# B&R Automation Studio project OpcUaSample410_BrbLibUa103 (part 10)

#### BrbUaAddNodeClassText.c - Gibt den Text einer NodeClass zurück
```c
#include <bur/plctypes.h>
#ifdef __cplusplus
	extern "C"
	{
#endif

#include "BrbLibUa.h"
#include <string.h>

#ifdef __cplusplus
	};
#endif

// NOLINTBEGIN(readability-*, bugprone-easily-swappable-parameters, bugprone-branch-clone, clang-diagnostic-invalid-utf8, clang-diagnostic-invalid-source-encoding, clang-diagnostic-pointer-arith, clang-diagnostic-strict-prototypes, hicpp-uppercase-literal-suffix, cppcoreguidelines-*, performance-*)

/* Hängt den Text einer NodeClass an */
plcdword BrbUaAddNodeClassText(enum UANodeClass eNodeClass, plcstring* pText, unsigned long nTextSize)
{
	DWORD nStatus = 0x80460000; // = Bad_StructureMissing
	if(pText != 0)
	{
		nStatus = 0x00000000; // = Good
		switch(eNodeClass)
		{
			case UANodeClass_None:
				BrbStringCat(pText, "None", nTextSize);
				break;

			case UANodeClass_Object:
				BrbStringCat(pText, "Object", nTextSize);
				break;

			case UANodeClass_Variable:
				BrbStringCat(pText, "Variable", nTextSize);
				break;

			case UANodeClass_Method:
				BrbStringCat(pText, "Method", nTextSize);
				break;

			case UANodeClass_ObjectType:
				BrbStringCat(pText, "ObjectType", nTextSize);
				break;

			case UANodeClass_VariableType:
				BrbStringCat(pText, "VariableType", nTextSize);
				break;

			case UANodeClass_ReferenceType:
				BrbStringCat(pText, "ReferenceType", nTextSize);
				break;

			case UANodeClass_DataType:
				BrbStringCat(pText, "DataType", nTextSize);
				break;

			case UANodeClass_View:
				BrbStringCat(pText, "View", nTextSize);
				break;

			case UANodeClass_All:
				BrbStringCat(pText, "All", nTextSize);
				break;

			default: // NOLINT(clang-diagnostic-covered-switch-default)
				BrbStringCat(pText, "Unknown", nTextSize);
				break;

		}
	}
	return nStatus;
}

// NOLINTEND(readability-*, bugprone-easily-swappable-parameters, bugprone-branch-clone, clang-diagnostic-invalid-utf8, clang-diagnostic-invalid-source-encoding, clang-diagnostic-pointer-arith, clang-diagnostic-strict-prototypes, hicpp-uppercase-literal-suffix, cppcoreguidelines-*, performance-*)
```

#### BrbUaAddDatatypeIdText.c - Gibt den Text zu einem Datentyp-Identifier zurück
```c
#include <bur/plctypes.h>
#ifdef __cplusplus
	extern "C"
	{
#endif

#include "BrbLibUa.h"
#include <string.h>

#ifdef __cplusplus
	};
#endif

// NOLINTBEGIN(readability-*, bugprone-easily-swappable-parameters, bugprone-branch-clone, clang-diagnostic-invalid-utf8, clang-diagnostic-invalid-source-encoding, clang-diagnostic-pointer-arith, clang-diagnostic-strict-prototypes, hicpp-uppercase-literal-suffix, cppcoreguidelines-*, performance-*)

/* Hängt den Text zu einem Datentyp-Identifier an */
plcdword BrbUaAddDatatypeIdText(unsigned long nDatatypeId, plcstring* pText, unsigned long nTextSize)
{
	DWORD nStatus = 0x80460000; // = Bad_StructureMissing
	if(pText != 0)
	{
		nStatus = 0x00000000; // = Good
		if(nDatatypeId == 1)
		{
			BrbStringCat(pText, "1=Boolean", nTextSize);
		}
		else if(nDatatypeId == 2)
		{
			BrbStringCat(pText, "2=SByte", nTextSize);
		}
		else if(nDatatypeId == 3)
		{
			BrbStringCat(pText, "3=Byte", nTextSize);
		}
		else if(nDatatypeId == 4)
		{
			BrbStringCat(pText, "4=Int16", nTextSize);
		}
		else if(nDatatypeId == 5)
		{
			BrbStringCat(pText, "5=UInt16", nTextSize);
		}
		else if(nDatatypeId == 6)
		{
			BrbStringCat(pText, "6=Int32", nTextSize);
		}
		else if(nDatatypeId == 7)
		{
			BrbStringCat(pText, "7=UInt32", nTextSize);
		}
		else if(nDatatypeId == 8)
		{
			BrbStringCat(pText, "8=Int64", nTextSize);
		}
		else if(nDatatypeId == 9)
		{
			BrbStringCat(pText, "9=UInt64", nTextSize);
		}
		else if(nDatatypeId == 10)
		{
			BrbStringCat(pText, "10=Float", nTextSize);
		}
		else if(nDatatypeId == 11)
		{
			BrbStringCat(pText, "11=Double", nTextSize);
		}
		else if(nDatatypeId == 12)
		{
			BrbStringCat(pText, "12=String", nTextSize);
		}
		else if(nDatatypeId == 13)
		{
			BrbStringCat(pText, "13=DateTime", nTextSize);
		}
		else if(nDatatypeId == 14)
		{
			BrbStringCat(pText, "14=Guid", nTextSize);
		}
		else if(nDatatypeId == 15)
		{
			BrbStringCat(pText, "15=ByteString", nTextSize);
		}
		else if(nDatatypeId == 16)
		{
			BrbStringCat(pText, "16=XmlElement", nTextSize);
		}
		else if(nDatatypeId == 17)
		{
			BrbStringCat(pText, "17=NodeId", nTextSize);
		}
		else if(nDatatypeId == 18)
		{
			BrbStringCat(pText, "18=ExpandedNodeId", nTextSize);
		}
		else if(nDatatypeId == 19)
		{
			BrbStringCat(pText, "19=StatusCode", nTextSize);
		}
		else if(nDatatypeId == 20)
		{
			BrbStringCat(pText, "20=QualifiedName", nTextSize);
		}
		else if(nDatatypeId == 21)
		{
			BrbStringCat(pText, "21=LocalizedText", nTextSize);
		}
		else if(nDatatypeId == 22)
		{
			BrbStringCat(pText, "22=Structure", nTextSize);
		}
		else if(nDatatypeId == 23)
		{
			BrbStringCat(pText, "23=DataValue", nTextSize);
		}
		else if(nDatatypeId == 25)
		{
			BrbStringCat(pText, "25=DiagnosticInfo", nTextSize);
		}
		else if(nDatatypeId == 26)
		{
			BrbStringCat(pText, "26=Number", nTextSize);
		}
		else if(nDatatypeId == 29)
		{
			BrbStringCat(pText, "29=Enumeration", nTextSize);
		}
		else if(nDatatypeId == 121)
		{
			BrbStringCat(pText, "121=Decimal128", nTextSize);
		}
		else
		{
			STRING sHelp[nBRBUA_VALUE_TEXT_CHAR_MAX];
			BrbUdintToAscii(nDatatypeId, sHelp);
			BrbStringCat(pText, sHelp, nTextSize);
		}
	}
	return nStatus;
}

// NOLINTEND(readability-*, bugprone-easily-swappable-parameters, bugprone-branch-clone, clang-diagnostic-invalid-utf8, clang-diagnostic-invalid-source-encoding, clang-diagnostic-pointer-arith, clang-diagnostic-strict-prototypes, hicpp-uppercase-literal-suffix, cppcoreguidelines-*, performance-*)
```

#### BrbUaAddArrayDimensionText.c - Gibt den Text für eine ArrayDimension zurück
```c
#include <bur/plctypes.h>
#ifdef __cplusplus
	extern "C"
	{
#endif

#include "BrbLibUa.h"
#include <string.h>

#ifdef __cplusplus
	};
#endif

// NOLINTBEGIN(readability-*, bugprone-easily-swappable-parameters, bugprone-branch-clone, clang-diagnostic-invalid-utf8, clang-diagnostic-invalid-source-encoding, clang-diagnostic-pointer-arith, clang-diagnostic-strict-prototypes, hicpp-uppercase-literal-suffix, cppcoreguidelines-*, performance-*)

/* Hängt den Text für eine ArrayDimension an */
plcdword BrbUaAddArrayDimensionText(unsigned long* pArrayDimension, signed long nValueRank, plcstring* pText, unsigned long nTextSize)
{
	DWORD nStatus = 0x80460000; // = Bad_StructureMissing
	if(pArrayDimension != 0 && pText != 0)
	{
		nStatus = 0x800F0000; // = Bad_NothingToDo
		if(nValueRank > 0)
		{
			nStatus = 0x00000000; // = Good
			DINT nIndex = 0;
			STRING sHelp[nBRBUA_VALUE_TEXT_CHAR_MAX];
			if(nValueRank > (DINT)MAX_ELEMENTS_ARRAYDIMENSION)
			{
				nValueRank = MAX_ELEMENTS_ARRAYDIMENSION;
			}
			for(nIndex=0; nIndex<=nValueRank-1; nIndex++)
			{
				UDINT* pDim = ((UDINT*)pArrayDimension) + nIndex;
				BrbUdintToAscii(*pDim, sHelp);
				BrbStringCat(pText, sHelp, nTextSize);
				BrbStringCat(pText, ";", nTextSize);
			}
			BrbStringTrimRight(pText, ";");
		}
	}
	return nStatus;
}

// NOLINTEND(readability-*, bugprone-easily-swappable-parameters, bugprone-branch-clone, clang-diagnostic-invalid-utf8, clang-diagnostic-invalid-source-encoding, clang-diagnostic-pointer-arith, clang-diagnostic-strict-prototypes, hicpp-uppercase-literal-suffix, cppcoreguidelines-*, performance-*)
```

#### BrbUaAddAccessLevelText.c - Gibt den Text eines AccessLevels zurück
```c
#include <bur/plctypes.h>
#ifdef __cplusplus
	extern "C"
	{
#endif

#include "BrbLibUa.h"
#include <string.h>

#ifdef __cplusplus
	};
#endif

// NOLINTBEGIN(readability-*, bugprone-easily-swappable-parameters, bugprone-branch-clone, clang-diagnostic-invalid-utf8, clang-diagnostic-invalid-source-encoding, clang-diagnostic-pointer-arith, clang-diagnostic-strict-prototypes, hicpp-uppercase-literal-suffix, cppcoreguidelines-*, performance-*)

/* Hängt den Text eines AccessLevels an */
plcdword BrbUaAddAccessLevelText(plcbyte nAccessLevel, plcstring* pText, unsigned long nTextSize)
{
	DWORD nStatus = 0x80460000; // = Bad_StructureMissing
	if(pText != 0)
	{
		nStatus = 0x00000000; // = Good
		STRING sHelp[nBRBUA_VALUE_TEXT_CHAR_MAX];
		brsitoa((DINT)nAccessLevel, (UDINT)&sHelp);
		BrbStringCat(pText, sHelp, nTextSize);
		BrbStringCat(pText, "=", nTextSize);
		if(nAccessLevel == 0)
		{
			BrbStringCat(pText, " None", nTextSize);
		}
		else
		{
			if(BrbGetBitUsint(nAccessLevel, 0) == 1)
			{
				BrbStringCat(pText, " Read,", nTextSize);
			}
			if(BrbGetBitUsint(nAccessLevel, 1) == 1)
			{
				BrbStringCat(pText, " Write,", nTextSize);
			}
			if(BrbGetBitUsint(nAccessLevel, 2) == 1)
			{
				BrbStringCat(pText, " HistoryRead,", nTextSize);
			}
			if(BrbGetBitUsint(nAccessLevel, 3) == 1)
			{
				BrbStringCat(pText, " HistoryWrite,", nTextSize);
			}
			BrbStringTrimLeft(pText, " ");
			BrbStringTrimRight(pText, " ");
			BrbStringTrimRight(pText, ",");
		}
	}
	return nStatus;
}

// NOLINTEND(readability-*, bugprone-easily-swappable-parameters, bugprone-branch-clone, clang-diagnostic-invalid-utf8, clang-diagnostic-invalid-source-encoding, clang-diagnostic-pointer-arith, clang-diagnostic-strict-prototypes, hicpp-uppercase-literal-suffix, cppcoreguidelines-*, performance-*)
```

#### BrbUaAddEventNotifierText.c - Gibt den Text eines EventNotifiers zurück
```c
#include <bur/plctypes.h>
#ifdef __cplusplus
	extern "C"
	{
#endif

#include "BrbLibUa.h"
#include <string.h>

#ifdef __cplusplus
	};
#endif

// NOLINTBEGIN(readability-*, bugprone-easily-swappable-parameters, bugprone-branch-clone, clang-diagnostic-invalid-utf8, clang-diagnostic-invalid-source-encoding, clang-diagnostic-pointer-arith, clang-diagnostic-strict-prototypes, hicpp-uppercase-literal-suffix, cppcoreguidelines-*, performance-*)

/* Hängt den Text eines EventNotifiers an */
plcdword BrbUaAddEventNotifierText(plcbyte nEventNotifier, plcstring* pText, unsigned long nTextSize)
{
	DWORD nStatus = 0x80460000; // = Bad_StructureMissing
	if(pText != 0)
	{
		nStatus = 0x00000000; // = Good
		STRING sHelp[nBRBUA_VALUE_TEXT_CHAR_MAX];
		brsitoa((DINT)nEventNotifier, (UDINT)&sHelp);
		BrbStringCat(pText, sHelp, nTextSize);
		BrbStringCat(pText, "=", nTextSize);
		if(nEventNotifier == 0)
		{
			BrbStringCat(pText, " None", nTextSize);
		}
		else
		{
			if(BrbGetBitUsint(nEventNotifier, 0) == 1)
			{
				BrbStringCat(pText, " Subscribe,", nTextSize);
			}
			if(BrbGetBitUsint(nEventNotifier, 2) == 1)
			{
				BrbStringCat(pText, " HistoryRead,", nTextSize);
			}
			if(BrbGetBitUsint(nEventNotifier, 3) == 1)
			{
				BrbStringCat(pText, " HistoryWrite,", nTextSize);
			}
			BrbStringTrimRight(pText, " ");
			BrbStringTrimLeft(pText, " ");
			BrbStringTrimRight(pText, ",");
		}
	}
	return nStatus;
}

// NOLINTEND(readability-*, bugprone-easily-swappable-parameters, bugprone-branch-clone, clang-diagnostic-invalid-utf8, clang-diagnostic-invalid-source-encoding, clang-diagnostic-pointer-arith, clang-diagnostic-strict-prototypes, hicpp-uppercase-literal-suffix, cppcoreguidelines-*, performance-*)
```

#### Package Logical/Libraries/BrbLibUa/General/VariantValues - Funktionen für OpcUa-Werte

#### BrbUaClearVariantValue.c
```c
#include <bur/plctypes.h>
#ifdef __cplusplus
	extern "C"
	{
#endif

#include "BrbLibUa.h"
#include <AnsiCFunc.h>
#include <string.h>

#ifdef __cplusplus
	};
#endif

// NOLINTBEGIN(readability-*, bugprone-easily-swappable-parameters, bugprone-branch-clone, clang-diagnostic-invalid-utf8, clang-diagnostic-invalid-source-encoding, clang-diagnostic-pointer-arith, clang-diagnostic-strict-prototypes, hicpp-uppercase-literal-suffix, cppcoreguidelines-*, performance-*)

/* Löscht den Inhalt eines OpcUa-Values, aber nicht die Datentyp-Angabe */
plcdword BrbUaClearVariantValue(struct UAVariantData* pUaVariantData)
{
	DWORD nStatus = 0x80460000; // = Bad_StructureMissing
	if(pUaVariantData != 0)
	{
		nStatus = 0x00000000; // = Good
		UAVariantType eVariantType = pUaVariantData->VariantType;
		memset(pUaVariantData, 0, sizeof(UAVariantData));
		pUaVariantData->VariantType = eVariantType;
	}
	return nStatus;
}

// NOLINTEND(readability-*, bugprone-easily-swappable-parameters, bugprone-branch-clone, clang-diagnostic-invalid-utf8, clang-diagnostic-invalid-source-encoding, clang-diagnostic-pointer-arith, clang-diagnostic-strict-prototypes, hicpp-uppercase-literal-suffix, cppcoreguidelines-*, performance-*)
```

#### BrbUaConvVariantValueFromString.c - Wandelt einen OpcUa-Value in einen Text
```c
#include <bur/plctypes.h>
#ifdef __cplusplus
	extern "C"
	{
#endif

#include "BrbLibUa.h"
#include <AnsiCFunc.h>
#include <string.h>

#ifdef __cplusplus
	};
#endif

// NOLINTBEGIN(readability-*, bugprone-easily-swappable-parameters, bugprone-branch-clone, clang-diagnostic-invalid-utf8, clang-diagnostic-invalid-source-encoding, clang-diagnostic-pointer-arith, clang-diagnostic-strict-prototypes, hicpp-uppercase-literal-suffix, cppcoreguidelines-*, performance-*)

/* Wandelt einen OpcUa-Value in einen Text */
plcdword BrbUaConvVariantValueFromString(struct UAVariantData* pUaVariantData, plcstring* pValueText)
{
	DWORD nStatus = 0x80460000; // = Bad_StructureMissing
	if(pUaVariantData != 0 && pValueText != 0)
	{
		nStatus = 0x00000000; // = Good
		// NOLINTBEGIN(bugprone-branch-clone)
		switch(pUaVariantData->VariantType)
		{
			case UAVariantType_Null:
				// Not supported by library
				BrbUaClearVariantValue(pUaVariantData);
				nStatus = 0x803D0000; // = Bad_NotSupported
				break;

			case UAVariantType_Boolean:
				BrbUaClearVariantValue(pUaVariantData);
				if(strcmp(pValueText, "True") == 0 || strcmp(pValueText, "true") == 0 || strcmp(pValueText, "1") == 0)
				{
					pUaVariantData->Boolean = 1;
				}
				else
				{
					pUaVariantData->Boolean = 0;
				}
				break;

			case UAVariantType_SByte:
				BrbUaClearVariantValue(pUaVariantData);
				pUaVariantData->SByte = (SINT)brsatoi((UDINT)pValueText);
				break;

			case UAVariantType_Byte:
				BrbUaClearVariantValue(pUaVariantData);
				pUaVariantData->Byte = (USINT)brsatoi((UDINT)pValueText);
				break;

			case UAVariantType_Int16:
				BrbUaClearVariantValue(pUaVariantData);
				pUaVariantData->Int16 = (INT)brsatoi((UDINT)pValueText);
				break;

			case UAVariantType_UInt16:
				BrbUaClearVariantValue(pUaVariantData);
				pUaVariantData->UInt16 = (UINT)brsatoi((UDINT)pValueText);
				break;

			case UAVariantType_Int32:
				BrbUaClearVariantValue(pUaVariantData);
				pUaVariantData->Int32 = brsatoi((UDINT)pValueText);
				break;

			case UAVariantType_UInt32:
				BrbUaClearVariantValue(pUaVariantData);
				pUaVariantData->UInt32 = BrbAsciiToUdint(pValueText);
				break;

			case UAVariantType_Int64:
				// No Element in structure
				BrbUaClearVariantValue(pUaVariantData);
				nStatus = 0x803D0000; // = Bad_NotSupported
				break;

			case UAVariantType_UInt64:
				// No Element in structure
				BrbUaClearVariantValue(pUaVariantData);
				nStatus = 0x803D0000; // = Bad_NotSupported
				break;

			case UAVariantType_Float:
				BrbUaClearVariantValue(pUaVariantData);
				BrbStringReplace(pValueText, ",", ".");
				pUaVariantData->Float = brsatof((UDINT)pValueText);
				break;

			case UAVariantType_Double:
				// Es gibt (noch) keine Umwandlungsfunktion von STRING auf LREAL
				// Deshalb wird zuerst in einen REAL gewandelt
				BrbUaClearVariantValue(pUaVariantData);
				BrbStringReplace(pValueText, ",", ".");
				pUaVariantData->Double = (LREAL)brsatof((UDINT)pValueText);
				break;

			case UAVariantType_String:
				BrbUaClearVariantValue(pUaVariantData);
				BrbStringCopy(pUaVariantData->String, pValueText, sizeof(pUaVariantData->String));
				break;

			case UAVariantType_DateTime:
				BrbUaClearVariantValue(pUaVariantData);
				pUaVariantData->DateTime = BrbGetDtFromTimeText(pValueText, sBRBUA_DATETIME_FORMAT);
				break;

			case UAVariantType_Guid:
				// Guid wird im String-Element gesetzt
				BrbUaClearVariantValue(pUaVariantData);
				BrbStringCopy(pUaVariantData->String, pValueText, sizeof(pUaVariantData->String));
				break;

			case UAVariantType_ByteString:
				// Not supported by library
				BrbUaClearVariantValue(pUaVariantData);
				nStatus = 0x803D0000; // = Bad_NotSupported
				break;

			case UAVariantType_XmlElement:
				// Not supported by library
				BrbUaClearVariantValue(pUaVariantData);
				nStatus = 0x803D0000; // = Bad_NotSupported
				break;

			case UAVariantType_NodeId:
				BrbUaClearVariantValue(pUaVariantData);
				pUaVariantData->NodeId.NamespaceIndex = 0;
				UDINT nTextLen = brsstrlen((UDINT)pValueText);
				DINT nEndCharIndexNs = 0;
				// NamespaceIndex
				if(BrbStringStartsWith(pValueText, "ns=") == 1)
				{
					nEndCharIndexNs = BrbStringGetIndexOf(pValueText, ";", nTextLen);
					if(nEndCharIndexNs > 3)
					{
						STRING sNamespaceIndex[32];
						BrbStringGetSubText((STRING*)pValueText, 3, (UDINT)nEndCharIndexNs-3, sNamespaceIndex);
						pUaVariantData->NodeId.NamespaceIndex = (UINT)brsatoi((UDINT)&sNamespaceIndex);
					}
					else if(nEndCharIndexNs == -1)
					{
						// Nur NamespaceIndex
						nEndCharIndexNs = (DINT)nTextLen-1;
						STRING sNamespaceIndex[32];
						BrbStringGetSubText((STRING*)pValueText, 3, (UDINT)nEndCharIndexNs-2, sNamespaceIndex);
						pUaVariantData->NodeId.NamespaceIndex = (UINT)brsatoi((UDINT)&sNamespaceIndex);
					}
				}
				// Identifier
				DINT nEndCharIndexId = (DINT)nTextLen-1;
				DINT nStartCharIndexId = BrbStringGetIndexOf(pValueText + nEndCharIndexNs, "i=", nTextLen);
				if(nStartCharIndexId > -1 && nEndCharIndexId > nStartCharIndexId+2)
				{
					pUaVariantData->NodeId.IdentifierType = UAIdentifierType_Numeric;
					STRING sIdentifier[255];
					nStartCharIndexId += 2;
					BrbStringGetSubText((STRING*)pValueText + nEndCharIndexNs, (UDINT)nStartCharIndexId, (UDINT)(nEndCharIndexId-nStartCharIndexId+1), sIdentifier);
					BrbStringCopy(pUaVariantData->NodeId.Identifier, sIdentifier, sizeof(pUaVariantData->NodeId.Identifier));
				}
				else
				{
					nStartCharIndexId = BrbStringGetIndexOf(pValueText + nEndCharIndexNs, "s=", nTextLen);
					if(nStartCharIndexId > -1 && nEndCharIndexId > nStartCharIndexId+2)
					{
						pUaVariantData->NodeId.IdentifierType = UAIdentifierType_String;
						STRING sIdentifier[255];
						nStartCharIndexId += 2;
						BrbStringGetSubText((STRING*)pValueText + nEndCharIndexNs, (UDINT)nStartCharIndexId, (UDINT)(nEndCharIndexId-nStartCharIndexId+1), sIdentifier);
						BrbStringCopy(pUaVariantData->NodeId.Identifier, sIdentifier, sizeof(pUaVariantData->NodeId.Identifier));
					}
					else
					{
						nStartCharIndexId = BrbStringGetIndexOf(pValueText + nEndCharIndexNs, "g=", nTextLen);
						if(nStartCharIndexId > -1 && nEndCharIndexId > nStartCharIndexId+2)
						{
							pUaVariantData->NodeId.IdentifierType = UAIdentifierType_GUID;
							STRING sIdentifier[255];
							nStartCharIndexId += 2;
							BrbStringGetSubText((STRING*)pValueText + nEndCharIndexNs, (UDINT)nStartCharIndexId, (UDINT)(nEndCharIndexId-nStartCharIndexId+1), sIdentifier);
							BrbStringCopy(pUaVariantData->NodeId.Identifier, sIdentifier, sizeof(pUaVariantData->NodeId.Identifier));
						}
					}
				}
				if(nStartCharIndexId == -1)
				{
					// Kein gültiger Identifier
					nStatus = 0x80330000 ; // = Bad_NodeIdInvalid
				}
				break;

			case UAVariantType_ExpandedNodeId:
				// Not supported by library
				BrbUaClearVariantValue(pUaVariantData);
				nStatus = 0x803D0000; // = Bad_NotSupported
				break;

			case UAVariantType_StatusCode:
				BrbUaClearVariantValue(pUaVariantData);
				if(BrbStringStartsWith(pValueText, "0x") == 1)
				{
					pUaVariantData->UInt32 = BrbHexToUdint(pValueText+2);
				}
				else
				{
					pUaVariantData->UInt32 = BrbAsciiToUdint(pValueText);
				}
				break;

			case UAVariantType_QualifiedName:
				// Not supported by library
				BrbUaClearVariantValue(pUaVariantData);
				nStatus = 0x803D0000; // = Bad_NotSupported
				break;

			case UAVariantType_LocalizedText:
				// Not supported by library
				BrbUaClearVariantValue(pUaVariantData);
				nStatus = 0x803D0000; // = Bad_NotSupported
				break;

		}
		// NOLINTEND(bugprone-branch-clone)
	}
	return nStatus;
}

// NOLINTEND(readability-*, bugprone-easily-swappable-parameters, bugprone-branch-clone, clang-diagnostic-invalid-utf8, clang-diagnostic-invalid-source-encoding, clang-diagnostic-pointer-arith, clang-diagnostic-strict-prototypes, hicpp-uppercase-literal-suffix, cppcoreguidelines-*, performance-*)
```

#### BrbUaConvVariantValueToString.c - Wandelt einen Text in einen OpcUa-Value
```c
#include <bur/plctypes.h>
#ifdef __cplusplus
	extern "C"
	{
#endif

#include "BrbLibUa.h"
#include <AnsiCFunc.h>
#include <string.h>

#ifdef __cplusplus
	};
#endif

// NOLINTBEGIN(readability-*, bugprone-easily-swappable-parameters, bugprone-branch-clone, clang-diagnostic-invalid-utf8, clang-diagnostic-invalid-source-encoding, clang-diagnostic-pointer-arith, clang-diagnostic-strict-prototypes, hicpp-uppercase-literal-suffix, cppcoreguidelines-*, performance-*)

/* Wandelt einen Text in einen OpcUa-Value */
plcdword BrbUaConvVariantValueToString(struct UAVariantData* pUaVariantData, plcstring* pValueText, unsigned long nValueTextSize)
{
	DWORD nStatus = 0x80460000; // = Bad_StructureMissing
	if(pUaVariantData != 0 && pValueText != 0)
	{
		nStatus = 0x00000000; // = Good
		STRING sHelp[255];
		memset(pValueText, 0, nValueTextSize);
		switch(pUaVariantData->VariantType)
		{
			case UAVariantType_Null:
				BrbStringCopy(pValueText, "Null", nValueTextSize);
				break;

			case UAVariantType_Boolean:
				if(pUaVariantData->Boolean == 1)
				{
					BrbStringCopy(pValueText, "True", nValueTextSize);
				}
				else
				{
					BrbStringCopy(pValueText, "False", nValueTextSize);
				}
				break;

			case UAVariantType_SByte:
				brsitoa((DINT)pUaVariantData->SByte, (UDINT)pValueText);
				break;

			case UAVariantType_Byte:
				brsitoa((DINT)pUaVariantData->Byte, (UDINT)pValueText);
				break;

			case UAVariantType_Int16:
				brsitoa((DINT)pUaVariantData->Int16, (UDINT)pValueText);
				break;

			case UAVariantType_UInt16:
				brsitoa((DINT)pUaVariantData->UInt16, (UDINT)pValueText);
				break;

			case UAVariantType_Int32:
				brsitoa((DINT)pUaVariantData->Int32, (UDINT)pValueText);
				break;

			case UAVariantType_UInt32:
				BrbUdintToAscii(pUaVariantData->UInt32, pValueText);
				break;

			case UAVariantType_Int64:
				BrbStringCopy(pValueText, "Int64 not supported!", nValueTextSize);
				nStatus = 0x803D0000; // = Bad_NotSupported
				break;

			case UAVariantType_UInt64:
				BrbStringCopy(pValueText, "UInt64 not supported!", nValueTextSize);
				nStatus = 0x803D0000; // = Bad_NotSupported
				break;

			case UAVariantType_Float:
				brsftoa(pUaVariantData->Float, (UDINT)pValueText);
				break;

			case UAVariantType_Double:
				// Es gibt (noch) keine Umwandlungsfunktion von LREAL auf STRING
				// Deshalb wird zuerst in einen REAL gewandelt
				brsftoa((REAL)pUaVariantData->Double, (UDINT)pValueText);
				break;

			case UAVariantType_String:
				BrbStringCopy(pValueText, pUaVariantData->String, nValueTextSize);
				break;

			case UAVariantType_DateTime:
				BrbGetTimeTextDt(pUaVariantData->DateTime, pValueText, nValueTextSize, sBRBUA_TIMESTAMP_FORMAT);
				break;

			case UAVariantType_Guid:
				BrbStringCopy(pValueText, pUaVariantData->String, nValueTextSize);
				break;

			case UAVariantType_ByteString:
				BrbStringCopy(pValueText, "Conversion of ByteString not supported!", nValueTextSize);
				nStatus = 0x803D0000; // = Bad_NotSupported
				break;

			case UAVariantType_XmlElement:
				BrbStringCopy(pValueText, "Conversion of XmlElement not supported!", nValueTextSize);
				nStatus = 0x803D0000; // = Bad_NotSupported
				break;

			case UAVariantType_NodeId:
				if(pUaVariantData->NodeId.IdentifierType == UAIdentifierType_String)
				{
					BrbStringCopy(pValueText, "ns=", nValueTextSize);
					brsitoa((DINT)pUaVariantData->NodeId.NamespaceIndex, (UDINT)&sHelp);
					BrbStringCat(pValueText, sHelp, nValueTextSize);
					BrbStringCat(pValueText, ";s=", nValueTextSize);
					BrbStringCat(pValueText, pUaVariantData->NodeId.Identifier, nValueTextSize);
				}
				else if(pUaVariantData->NodeId.IdentifierType == UAIdentifierType_Numeric)
				{
					BrbStringCopy(pValueText, "ns=", nValueTextSize);
					brsitoa((DINT)pUaVariantData->NodeId.NamespaceIndex, (UDINT)&sHelp);
					BrbStringCat(pValueText, sHelp, nValueTextSize);
					BrbStringCat(pValueText, ";i=", nValueTextSize);
					BrbStringCat(pValueText, pUaVariantData->NodeId.Identifier, nValueTextSize);
				}
				else if(pUaVariantData->NodeId.IdentifierType == UAIdentifierType_GUID)
				{
					BrbStringCopy(pValueText, "ns=", nValueTextSize);
					brsitoa((DINT)pUaVariantData->NodeId.NamespaceIndex, (UDINT)&sHelp);
					BrbStringCat(pValueText, sHelp, nValueTextSize);
					BrbStringCat(pValueText, ";g=", nValueTextSize);
					BrbStringCat(pValueText, pUaVariantData->NodeId.Identifier, nValueTextSize);
				}
				else if(pUaVariantData->NodeId.IdentifierType == UAIdentifierType_Opaque)
				{
					BrbStringCopy(pValueText, "Conversion of opaque node id not supported!", nValueTextSize);
					nStatus = 0x803D0000; // = Bad_NotSupported
				}
				break;

			case UAVariantType_ExpandedNodeId:
				BrbStringCopy(pValueText, "Conversion of expanded node id not supported!", nValueTextSize);
				nStatus = 0x803D0000; // = Bad_NotSupported
				break;

			case UAVariantType_StatusCode:
				BrbUaGetStatusCodeText(pUaVariantData->UInt32, pValueText, nValueTextSize);
				break;

			case UAVariantType_QualifiedName:
				brsitoa((DINT)pUaVariantData->QualifiedName.NamespaceIndex, (UDINT)pValueText);
				BrbStringCat(pValueText, ":", nValueTextSize);
				BrbStringCat(pValueText, pUaVariantData->QualifiedName.Name, nValueTextSize);
				break;

			case UAVariantType_LocalizedText:
				if(strlen(pUaVariantData->LocalizedText.Locale) > 0)
				{
					BrbStringCopy(pValueText, pUaVariantData->LocalizedText.Locale, nValueTextSize);
					BrbStringCat(pValueText, ":", nValueTextSize);
					BrbStringCat(pValueText, pUaVariantData->LocalizedText.Text, nValueTextSize);
				}
				else
				{
					BrbStringCopy(pValueText, pUaVariantData->LocalizedText.Text, nValueTextSize);
				}
				break;

		}
	}
	return nStatus;
}

// NOLINTEND(readability-*, bugprone-easily-swappable-parameters, bugprone-branch-clone, clang-diagnostic-invalid-utf8, clang-diagnostic-invalid-source-encoding, clang-diagnostic-pointer-arith, clang-diagnostic-strict-prototypes, hicpp-uppercase-literal-suffix, cppcoreguidelines-*, performance-*)
```

#### BrbUaAddVariantValueSubName.c - Hängt den Element-Namen eines OpcUa-Values anhand des Datentypen an einen Text an
```c
#include <bur/plctypes.h>
#ifdef __cplusplus
	extern "C"
	{
#endif

#include "BrbLibUa.h"
#include <AnsiCFunc.h>
#include <string.h>

#ifdef __cplusplus
	};
#endif

// NOLINTBEGIN(readability-*, bugprone-easily-swappable-parameters, bugprone-branch-clone, clang-diagnostic-invalid-utf8, clang-diagnostic-invalid-source-encoding, clang-diagnostic-pointer-arith, clang-diagnostic-strict-prototypes, hicpp-uppercase-literal-suffix, cppcoreguidelines-*, performance-*)

/* Hängt den Element-Namen eines OpcUa-Values anhand des Datentypen an einen Text an */
plcdword BrbUaAddVariantValueSubName(enum UAVariantType eVariantType, plcstring* pText, unsigned long nTextSize)
{
	DWORD nStatus = 0x80460000; // = Bad_StructureMissing
	if(pText != 0)
	{
		nStatus = 0x00000000; // = Good
		// NOLINTBEGIN(bugprone-branch-clone)
		switch(eVariantType) // NOLINT(hicpp-multiway-paths-covered)
		{
			case UAVariantType_Null:
				// Not supported
				nStatus = 0x803D0000; // = Bad_NotSupported
				break;

			case UAVariantType_Boolean:
				BrbStringCat(pText, ".Boolean", nTextSize);
				break;

			case UAVariantType_SByte:
				BrbStringCat(pText, ".SByte", nTextSize);
				break;

			case UAVariantType_Byte:
				BrbStringCat(pText, ".Byte", nTextSize);
				break;

			case UAVariantType_Int16:
				BrbStringCat(pText, ".Int16", nTextSize);
				break;

			case UAVariantType_UInt16:
				BrbStringCat(pText, ".UInt16", nTextSize);
				break;

			case UAVariantType_Int32:
				BrbStringCat(pText, ".Int32", nTextSize);
				break;

			case UAVariantType_UInt32:
				BrbStringCat(pText, ".UInt32", nTextSize);
				break;

			case UAVariantType_Int64:
				BrbStringCat(pText, ".Int64", nTextSize);
				break;

			case UAVariantType_UInt64:
				BrbStringCat(pText, ".UInt64", nTextSize);
				break;

			case UAVariantType_Float:
				BrbStringCat(pText, ".Float", nTextSize);
				break;

			case UAVariantType_Double:
				BrbStringCat(pText, ".Double", nTextSize);
				break;

			case UAVariantType_String:
				BrbStringCat(pText, ".String", nTextSize);
				break;

			case UAVariantType_DateTime:
				BrbStringCat(pText, ".DateTime", nTextSize);
				break;

			case UAVariantType_Guid:
				BrbStringCat(pText, ".String", nTextSize);
				break;

			case UAVariantType_ByteString:
				BrbStringCat(pText, ".String", nTextSize);
				break;

			case UAVariantType_XmlElement:
				// Not supported
				nStatus = 0x803D0000; // = Bad_NotSupported
				break;

			case UAVariantType_NodeId:
				BrbStringCat(pText, ".NodeId", nTextSize);
				break;

			case UAVariantType_ExpandedNodeId:
				BrbStringCat(pText, ".ExpandedNodeId", nTextSize);
				break;

			case UAVariantType_StatusCode:
				BrbStringCat(pText, ".StatusCode", nTextSize);
				break;

			case UAVariantType_QualifiedName:
				BrbStringCat(pText, ".QualifiedName", nTextSize);
				break;

			case UAVariantType_LocalizedText:
				BrbStringCat(pText, ".LocalizedText", nTextSize);
				break;

		}
		// NOLINTEND(bugprone-branch-clone)
	}
	return nStatus;
}

// NOLINTEND(readability-*, bugprone-easily-swappable-parameters, bugprone-branch-clone, clang-diagnostic-invalid-utf8, clang-diagnostic-invalid-source-encoding, clang-diagnostic-pointer-arith, clang-diagnostic-strict-prototypes, hicpp-uppercase-literal-suffix, cppcoreguidelines-*, performance-*)
```

#### Package Logical/Libraries/BrbLibUa/General/ByteStrings - Funktionen für OpcUa-Ereignisse

#### BrbUaIncByteString.c
```c
#include <bur/plctypes.h>
#ifdef __cplusplus
	extern "C"
	{
#endif

#include "BrbLibUa.h"
#include <AnsiCFunc.h>
#include <string.h>

#ifdef __cplusplus
	};
#endif

// NOLINTBEGIN(readability-*, bugprone-easily-swappable-parameters, bugprone-branch-clone, clang-diagnostic-invalid-utf8, clang-diagnostic-invalid-source-encoding, clang-diagnostic-pointer-arith, clang-diagnostic-strict-prototypes, hicpp-uppercase-literal-suffix, cppcoreguidelines-*, performance-*)

/* Inkrementiert einen ByteString */
plcdword BrbUaIncByteString(unsigned char* pData, signed long nLength)
{
	DWORD nStatus = 0x80460000; // = Bad_StructureMissing
	if(pData != 0)
	{
		nStatus = 0x803C0000; // = Bad_OutOfRange
		if(nLength > 0)
		{
			nStatus = 0x00000000; // = Good
			DINT nIndex = nLength - 1;
			BOOL bLeave = 0;
			do
			{
				USINT* pValue = (USINT*)pData + nIndex;
				if(*pValue < 255)
				{
					*pValue += 1;
					bLeave = 1;
				}
				else
				{
					*pValue = 0;
					nIndex -= 1;
					if(nIndex < 0)
					{
						// Überlauf -> Wieder bei 0 beginnen
						memset(pData, 0, (UDINT)nLength);
						nStatus = 0xB00C0000; // = PlcOpen_BadElementCount
						bLeave = 1;
					}
				}
			} while (bLeave == 0);
		}
	}
	return nStatus;
}

// NOLINTEND(readability-*, bugprone-easily-swappable-parameters, bugprone-branch-clone, clang-diagnostic-invalid-utf8, clang-diagnostic-invalid-source-encoding, clang-diagnostic-pointer-arith, clang-diagnostic-strict-prototypes, hicpp-uppercase-literal-suffix, cppcoreguidelines-*, performance-*)
```

#### BrbUaGetRandomByteString.c
```c
#include <bur/plctypes.h>
#ifdef __cplusplus
	extern "C"
	{
#endif

#include "BrbLibUa.h"
#include <string.h>

#ifdef __cplusplus
	};
#endif

// NOLINTBEGIN(readability-*, bugprone-easily-swappable-parameters, bugprone-branch-clone, clang-diagnostic-invalid-utf8, clang-diagnostic-invalid-source-encoding, clang-diagnostic-pointer-arith, clang-diagnostic-strict-prototypes, hicpp-uppercase-literal-suffix, cppcoreguidelines-*, performance-*)

/* Erzeugt einen zufälligen ByteString */
plcdword BrbUaGetRandomByteString(unsigned char* pData, signed long nLength)
{
	DWORD nStatus = 0x80460000; // = Bad_StructureMissing
	if(pData != 0)
	{
		nStatus = 0x803C0000; // = Bad_OutOfRange
		if(nLength > 0)
		{
			nStatus = 0x00000000; // = Good
			DINT nIndex = 0;
			for(nIndex=0; nIndex<nLength; nIndex++)
			{
				*(pData + nIndex) = (USINT)BrbGetRandomDint(0, 255);
			}
		}
	}
	return nStatus;
}

// NOLINTEND(readability-*, bugprone-easily-swappable-parameters, bugprone-branch-clone, clang-diagnostic-invalid-utf8, clang-diagnostic-invalid-source-encoding, clang-diagnostic-pointer-arith, clang-diagnostic-strict-prototypes, hicpp-uppercase-literal-suffix, cppcoreguidelines-*, performance-*)
```

#### BrbUaLoadImage.c
```c
#include <bur/plctypes.h>
#ifdef __cplusplus
	extern "C"
	{
#endif

#include "BrbLibUa.h"
#include <string.h>
#include <AnsiCFunc.h>

#ifdef __cplusplus
	};
#endif

// NOLINTBEGIN(readability-*, bugprone-easily-swappable-parameters, bugprone-branch-clone, clang-diagnostic-invalid-utf8, clang-diagnostic-invalid-source-encoding, clang-diagnostic-pointer-arith, clang-diagnostic-strict-prototypes, hicpp-uppercase-literal-suffix, cppcoreguidelines-*, performance-*)

// Eigene Enums und Typen
enum Steps_ENUM
{
	eSTEP_INIT,
	eSTEP_LOAD_FILE,
	eSTEP_LOAD_FILE_WAT,
};

/* Lädt ein Image */
void BrbUaLoadImage(struct BrbUaLoadImage* inst)
{
	switch(inst->eStep)
	{
		case eSTEP_INIT:
			// Fub initialisieren
			inst->nStatus =  65535;
			if(inst->pDevice != 0 && inst->pFile != 0 && inst->pImageData != 0 && inst->pImageLength != 0)
			{
				memset(&inst->fbBrbLoadFileBin, 0, sizeof(inst->fbBrbLoadFileBin));
				inst->eStep = eSTEP_LOAD_FILE;
			}
			else
			{
				inst->nStatus = eBRB_ERR_NULL_POINTER;
			}
			break;

		case eSTEP_LOAD_FILE:
			// Datei laden
			inst->nStatus  = eBRB_ERR_BUSY;
			inst->fbBrbLoadFileBin.pDevice = (STRING*)inst->pDevice;
			inst->fbBrbLoadFileBin.pFile = (STRING*)inst->pFile;
			inst->fbBrbLoadFileBin.pVar = (USINT*)inst->pImageData;
			inst->fbBrbLoadFileBin.nVarSize = inst->nImageDataSize;
			inst->eStep = eSTEP_LOAD_FILE_WAT;
			break;

		case eSTEP_LOAD_FILE_WAT:
			// Warten, bis Datei geladen ist
			BrbLoadFileBin(&inst->fbBrbLoadFileBin);
			if(inst->fbBrbLoadFileBin.nStatus == 0)
			{
				inst->nStatus = inst->fbBrbLoadFileBin.nStatus;
				*inst->pImageLength = (DINT)inst->fbBrbLoadFileBin.nValidBytes;
				inst->eStep = eSTEP_INIT;
			}
			else if(inst->fbBrbLoadFileBin.nStatus != 65535)
			{
				inst->nStatus = inst->fbBrbLoadFileBin.nStatus;
				*inst->pImageLength = 0;
				inst->eStep = eSTEP_INIT;
			}
			break;

	}
}

// NOLINTEND(readability-*, bugprone-easily-swappable-parameters, bugprone-branch-clone, clang-diagnostic-invalid-utf8, clang-diagnostic-invalid-source-encoding, clang-diagnostic-pointer-arith, clang-diagnostic-strict-prototypes, hicpp-uppercase-literal-suffix, cppcoreguidelines-*, performance-*)
```

#### BrbUaSetLocalizedText.c
```c
#include <bur/plctypes.h>
#ifdef __cplusplus
	extern "C"
	{
#endif

#include "BrbLibUa.h"
#include <string.h>

#ifdef __cplusplus
	};
#endif

// NOLINTBEGIN(readability-*, bugprone-easily-swappable-parameters, bugprone-branch-clone, clang-diagnostic-invalid-utf8, clang-diagnostic-invalid-source-encoding, clang-diagnostic-pointer-arith, clang-diagnostic-strict-prototypes, hicpp-uppercase-literal-suffix, cppcoreguidelines-*, performance-*)

/* Besetzt einen LocalizedText */
plcdword BrbUaSetLocalizedText(BrUaLocalizedText* pLocalizedText, plcstring* pLocale, plcstring* pText)
{
	DWORD nStatus = 0x80460000; // = Bad_StructureMissing
	if(pLocalizedText != 0 && pLocale != 0 && pText != 0)
	{
		nStatus = 0x00000000; // = Good
		BrbStringCopy(pLocalizedText->Locale, pLocale, sizeof(pLocalizedText->Locale));
		BrbStringCopy(pLocalizedText->Text, pText, sizeof(pLocalizedText->Text));
	}
	return nStatus;
}

// NOLINTEND(readability-*, bugprone-easily-swappable-parameters, bugprone-branch-clone, clang-diagnostic-invalid-utf8, clang-diagnostic-invalid-source-encoding, clang-diagnostic-pointer-arith, clang-diagnostic-strict-prototypes, hicpp-uppercase-literal-suffix, cppcoreguidelines-*, performance-*)
```

#### BrbUaGetRandomLocalizedText.c
```c
#include <bur/plctypes.h>
#ifdef __cplusplus
	extern "C"
	{
#endif

#include "BrbLibUa.h"
#include <string.h>

#ifdef __cplusplus
	};
#endif

// NOLINTBEGIN(readability-*, bugprone-easily-swappable-parameters, bugprone-branch-clone, clang-diagnostic-invalid-utf8, clang-diagnostic-invalid-source-encoding, clang-diagnostic-pointer-arith, clang-diagnostic-strict-prototypes, hicpp-uppercase-literal-suffix, cppcoreguidelines-*, performance-*)

/* Erezugt einen zufälligen LocalizedText */
plcdword BrbUaGetRandomLocalizedText(BrUaLocalizedText* pLocalizedText, unsigned short nLength)
{
	DWORD nStatus = 0x80460000; // = Bad_StructureMissing
	if(pLocalizedText != 0)
	{
		nStatus = 0x00000000; // = Good
		STRING sLocale[6];
		UINT nLocale = (UINT)BrbGetRandomUdint(0,3);
		if(nLocale == 0)
		{
			BrbStringCopy(sLocale, "de", sizeof(sLocale));
		}
		else if(nLocale == 1)
		{
			BrbStringCopy(sLocale, "en", sizeof(sLocale));
		}
		else if(nLocale == 2)
		{
			BrbStringCopy(sLocale, "fr", sizeof(sLocale));
		}
		else if(nLocale == 3)
		{
			BrbStringCopy(sLocale, "es", sizeof(sLocale));
		}
		if(nLength > 255)
		{
			nLength = 255;
		}
		STRING sText[255];
		BrbGetRandomText((STRING*)&sText, sizeof(sText), nLength);
		BrbUaSetLocalizedText(pLocalizedText, sLocale, sText);
	}
	return nStatus;
}

// NOLINTEND(readability-*, bugprone-easily-swappable-parameters, bugprone-branch-clone, clang-diagnostic-invalid-utf8, clang-diagnostic-invalid-source-encoding, clang-diagnostic-pointer-arith, clang-diagnostic-strict-prototypes, hicpp-uppercase-literal-suffix, cppcoreguidelines-*, performance-*)
```

#### BrbUaAddLocalizedTextText.c
```c
#include <bur/plctypes.h>
#ifdef __cplusplus
	extern "C"
	{
#endif

#include "BrbLibUa.h"
#include <string.h>

#ifdef __cplusplus
	};
#endif

// NOLINTBEGIN(readability-*, bugprone-easily-swappable-parameters, bugprone-branch-clone, clang-diagnostic-invalid-utf8, clang-diagnostic-invalid-source-encoding, clang-diagnostic-pointer-arith, clang-diagnostic-strict-prototypes, hicpp-uppercase-literal-suffix, cppcoreguidelines-*, performance-*)

/* Hängt den Text eines LocalizedText an */
plcdword BrbUaAddLocalizedTextText(BrUaLocalizedText* pLocalizedText, plcstring* pText, unsigned long nTextSize)
{
	DWORD nStatus = 0x80460000; // = Bad_StructureMissing
	if(pLocalizedText != 0 && pText != 0)
	{
		nStatus = 0x00000000; // = Good
		if(strlen(pLocalizedText->Locale) > 0)
		{
			BrbStringCat(pText, pLocalizedText->Locale, nTextSize);
			BrbStringCat(pText, ":", nTextSize);
		}
		BrbStringCat(pText, pLocalizedText->Text, nTextSize);
	}
	return nStatus;
}

// NOLINTEND(readability-*, bugprone-easily-swappable-parameters, bugprone-branch-clone, clang-diagnostic-invalid-utf8, clang-diagnostic-invalid-source-encoding, clang-diagnostic-pointer-arith, clang-diagnostic-strict-prototypes, hicpp-uppercase-literal-suffix, cppcoreguidelines-*, performance-*)
```

#### BrbUaSetQualifedName.c
```c
#include <bur/plctypes.h>
#ifdef __cplusplus
	extern "C"
	{
#endif

#include "BrbLibUa.h"
#include <string.h>

#ifdef __cplusplus
	};
#endif

// NOLINTBEGIN(readability-*, bugprone-easily-swappable-parameters, bugprone-branch-clone, clang-diagnostic-invalid-utf8, clang-diagnostic-invalid-source-encoding, clang-diagnostic-pointer-arith, clang-diagnostic-strict-prototypes, hicpp-uppercase-literal-suffix, cppcoreguidelines-*, performance-*)

/* Besetzt einen QualifiedName */
plcdword BrbUaSetQualifedName(BrUaQualifiedName* pQualifiedName, unsigned short nNamespaceIndex, plcstring* pName)
{
	DWORD nStatus = 0x80460000; // = Bad_StructureMissing
	if(pQualifiedName != 0 && pName != 0)
	{
		nStatus = 0x00000000; // = Good
		pQualifiedName->NamespaceIndex = nNamespaceIndex;
		BrbStringCopy(pQualifiedName->Name, pName, sizeof(pQualifiedName->Name));
	}
	return nStatus;
}

// NOLINTEND(readability-*, bugprone-easily-swappable-parameters, bugprone-branch-clone, clang-diagnostic-invalid-utf8, clang-diagnostic-invalid-source-encoding, clang-diagnostic-pointer-arith, clang-diagnostic-strict-prototypes, hicpp-uppercase-literal-suffix, cppcoreguidelines-*, performance-*)
```

#### BrbUaGetRandomQualifiedName.c
```c
#include <bur/plctypes.h>
#ifdef __cplusplus
	extern "C"
	{
#endif

#include "BrbLibUa.h"
#include <string.h>

#ifdef __cplusplus
	};
#endif

// NOLINTBEGIN(readability-*, bugprone-easily-swappable-parameters, bugprone-branch-clone, clang-diagnostic-invalid-utf8, clang-diagnostic-invalid-source-encoding, clang-diagnostic-pointer-arith, clang-diagnostic-strict-prototypes, hicpp-uppercase-literal-suffix, cppcoreguidelines-*, performance-*)

/* Erzeugt einen zufälligen QualifiedName */
plcdword BrbUaGetRandomQualifiedName(BrUaQualifiedName* pQualifiedName, unsigned short nLength)
{
	DWORD nStatus = 0x80460000; // = Bad_StructureMissing
	if(pQualifiedName != 0)
	{
		nStatus = 0x00000000; // = Good
		UINT nNamespaceIndex = (UINT)BrbGetRandomUdint(0,65535);
		if(nLength > 255)
		{
			nLength = 255;
		}
		STRING sName[255];
		BrbGetRandomText((STRING*)&sName, sizeof(sName), nLength);
		BrbUaSetQualifedName(pQualifiedName, nNamespaceIndex, sName);
	}
	return nStatus;
}

// NOLINTEND(readability-*, bugprone-easily-swappable-parameters, bugprone-branch-clone, clang-diagnostic-invalid-utf8, clang-diagnostic-invalid-source-encoding, clang-diagnostic-pointer-arith, clang-diagnostic-strict-prototypes, hicpp-uppercase-literal-suffix, cppcoreguidelines-*, performance-*)
```

#### BrbUaDtStructToUaSrvDateTime.c
```c
#include <bur/plctypes.h>
#ifdef __cplusplus
	extern "C"
	{
#endif

#include "BrbLibUa.h"
#include <string.h>

#ifdef __cplusplus
	};
#endif

// NOLINTBEGIN(readability-*, bugprone-easily-swappable-parameters, bugprone-branch-clone, clang-diagnostic-invalid-utf8, clang-diagnostic-invalid-source-encoding, clang-diagnostic-pointer-arith, clang-diagnostic-strict-prototypes, hicpp-uppercase-literal-suffix, cppcoreguidelines-*, performance-*)

/* Wandelt eine DtStruct-Zeit in eine UaSrvDateTime-Zeit */
unsigned short BrbUaDtStructToUaSrvDateTime(struct UaSrv_DateTimeType* pUaSrvDateTime, struct DTStructure* pDtStruct, unsigned short nNanoSeconds)
{
	if(pUaSrvDateTime == 0)
	{
		return eBRB_ERR_NULL_POINTER;
	}
	if(pDtStruct == 0)
	{
		return eBRB_ERR_NULL_POINTER;
	}
	memset(pUaSrvDateTime, 0, sizeof(UaSrv_DateTimeType));
	pUaSrvDateTime->DateTime = DTStructure_TO_DT((UDINT)pDtStruct);
	pUaSrvDateTime->NanoSeconds = pDtStruct->millisec * 1000000 + pDtStruct->microsec * 1000 + nNanoSeconds;
	return eBRB_ERR_OK;
}

// NOLINTEND(readability-*, bugprone-easily-swappable-parameters, bugprone-branch-clone, clang-diagnostic-invalid-utf8, clang-diagnostic-invalid-source-encoding, clang-diagnostic-pointer-arith, clang-diagnostic-strict-prototypes, hicpp-uppercase-literal-suffix, cppcoreguidelines-*, performance-*)
```

#### BrbUaSrvDateTimeToDtStruct.c
```c
#include <bur/plctypes.h>
#ifdef __cplusplus
	extern "C"
	{
#endif

#include "BrbLibUa.h"
#include <string.h>

#ifdef __cplusplus
	};
#endif

// NOLINTBEGIN(readability-*, bugprone-easily-swappable-parameters, bugprone-branch-clone, clang-diagnostic-invalid-utf8, clang-diagnostic-invalid-source-encoding, clang-diagnostic-pointer-arith, clang-diagnostic-strict-prototypes, hicpp-uppercase-literal-suffix, cppcoreguidelines-*, performance-*)

/* Wandelt eine UaSrvDateTime-Zeit in eine DtStruct-Zeit */
unsigned short BrbUaSrvDateTimeToDtStruct(struct DTStructure* pDtStruct, struct UaSrv_DateTimeType* pUaSrvDateTime)
{
	if(pDtStruct == 0)
	{
		return eBRB_ERR_NULL_POINTER;
	}
	if(pUaSrvDateTime == 0)
	{
		return eBRB_ERR_NULL_POINTER;
	}
	memset(pDtStruct, 0, sizeof(DTStructure));
	DT_TO_DTStructure(pUaSrvDateTime->DateTime, (UDINT)pDtStruct);
	UDINT nTotalNanoSeconds = pUaSrvDateTime->NanoSeconds;
	pDtStruct->millisec = (UINT)(nTotalNanoSeconds / 1000000);
	nTotalNanoSeconds -= pDtStruct->millisec * 1000000;
	pDtStruct->microsec = (UINT)(nTotalNanoSeconds / 1000);
	BrbGetWeekdayDtStruct(pDtStruct);
	return eBRB_ERR_OK;
}

// NOLINTEND(readability-*, bugprone-easily-swappable-parameters, bugprone-branch-clone, clang-diagnostic-invalid-utf8, clang-diagnostic-invalid-source-encoding, clang-diagnostic-pointer-arith, clang-diagnostic-strict-prototypes, hicpp-uppercase-literal-suffix, cppcoreguidelines-*, performance-*)
```

#### BrbUaGetSrvTimeText.c
```c
#include <bur/plctypes.h>
#ifdef __cplusplus
	extern "C"
	{
#endif

#include "BrbLibUa.h"
#include <string.h>

#ifdef __cplusplus
	};
#endif

// NOLINTBEGIN(readability-*, bugprone-easily-swappable-parameters, bugprone-branch-clone, clang-diagnostic-invalid-utf8, clang-diagnostic-invalid-source-encoding, clang-diagnostic-pointer-arith, clang-diagnostic-strict-prototypes, hicpp-uppercase-literal-suffix, cppcoreguidelines-*, performance-*)

/* Gibt den Text eines Server-Zeitstempels zurück */
unsigned short BrbUaGetSrvTimeText(struct UaSrv_DateTimeType* pSrvTime, plcstring* pText, unsigned long nTextSize, signed short nTimeOffset, plcstring* pFormat)
{
	// Prüfung der Parameter
	if(pSrvTime == 0)
	{
		return eBRB_ERR_NULL_POINTER;
	}
	if(pText == 0)
	{
		return eBRB_ERR_NULL_POINTER;
	}
	if(nTextSize == 0)
	{
		return eBRB_ERR_INVALID_PARAMETER;
	}
	if(pFormat == 0)
	{
		return eBRB_ERR_NULL_POINTER;
	}
	// Zuerst die Werte umwandeln
	DTStructure DtStruct;
	DT_TO_DTStructure(pSrvTime->DateTime, (UDINT)&DtStruct);
	BrbDtStructAddMinutes(&DtStruct, nTimeOffset);
	UDINT nTotalNanoSeconds = pSrvTime->NanoSeconds;
	DtStruct.millisec = (UINT)(nTotalNanoSeconds / 1000000);
	nTotalNanoSeconds -= DtStruct.millisec * 1000000;
	DtStruct.microsec = (UINT)(nTotalNanoSeconds / 1000);
	nTotalNanoSeconds -= DtStruct.microsec * 1000;
	UINT nNanoSeconds = (UINT)nTotalNanoSeconds;
	// Alle Stellen werden mit führenden Nullen aufgefüllt
	memset((USINT*)pText, 0, nTextSize);
	BrbStringCopy(pText, pFormat, nTextSize);
	STRING sItoA[20];
	memset((USINT*)sItoA, 0, sizeof(sItoA));
	if(BrbStringGetAdrOf(pText, "mil", 0) != 0)
	{
		brsitoa((DINT)DtStruct.millisec, (UDINT)&sItoA);
		if(DtStruct.millisec < 10)
		{
			BrbStringInsert(sItoA, 0, "00");
		}
		else if(DtStruct.millisec < 100)
		{
			BrbStringInsert(sItoA, 0, "0");
		}
		BrbStringReplace(pText, "mil", sItoA);
	}
	if(BrbStringGetAdrOf(pText, "mic", 0) != 0)
	{
		brsitoa((DINT)DtStruct.microsec, (UDINT)&sItoA);
		if(DtStruct.microsec < 10)
		{
			BrbStringInsert(sItoA, 0, "00");
		}
		else if(DtStruct.microsec < 100)
		{
			BrbStringInsert(sItoA, 0, "0");
		}
		BrbStringReplace(pText, "mic", sItoA);
	}
	if(BrbStringGetAdrOf(pText, "nan", 0) != 0)
	{
		brsitoa((DINT)nNanoSeconds, (UDINT)&sItoA);
		if(nNanoSeconds < 10)
		{
			BrbStringInsert(sItoA, 0, "00");
		}
		else if(nNanoSeconds < 100)
		{
			BrbStringInsert(sItoA, 0, "0");
		}
		BrbStringReplace(pText, "nan", sItoA);
	}
	if(BrbStringGetAdrOf(pText, "yyyy", 0) != 0)
	{
		brsitoa((DINT)DtStruct.year, (UDINT)&sItoA);
		BrbStringPadLeft(sItoA, "0", 4);
		BrbStringReplace(pText, "yyyy", sItoA);
	}
	else if(BrbStringGetAdrOf(pText, "yy", 0) != 0)
	{
		DtStruct.year -= 2000;
		brsitoa((DINT)DtStruct.year, (UDINT)&sItoA);
		BrbStringPadLeft(sItoA, "0", 2);
		BrbStringReplace(pText, "yy", sItoA);
	}
	if(BrbStringGetAdrOf(pText, "mm", 0) != 0)
	{
		brsitoa((DINT)DtStruct.month, (UDINT)&sItoA);
		if(DtStruct.month < 10)
		{
			BrbStringInsert(sItoA, 0, "0");
		}
		BrbStringReplace(pText, "mm", sItoA);
	}
	else if(BrbStringGetAdrOf(pText, "m", 0) != 0)
	{
		brsitoa((DINT)DtStruct.month, (UDINT)&sItoA);
		BrbStringReplace(pText, "m", sItoA);
	}
	if(BrbStringGetAdrOf(pText, "dd", 0) != 0)
	{
		brsitoa((DINT)DtStruct.day, (UDINT)&sItoA);
		if(DtStruct.day < 10)
		{
			BrbStringInsert(sItoA, 0, "0");
		}
		BrbStringReplace(pText, "dd", sItoA);
	}
	else if(BrbStringGetAdrOf(pText, "d", 0) != 0)
	{
		brsitoa((DINT)DtStruct.day, (UDINT)&sItoA);
		BrbStringReplace(pText, "d", sItoA);
	}
	if(BrbStringGetAdrOf(pText, "hh", 0) != 0)
	{
		brsitoa((DINT)DtStruct.hour, (UDINT)&sItoA);
		if(DtStruct.hour < 10)
		{
			BrbStringInsert(sItoA, 0, "0");
		}
		BrbStringReplace(pText, "hh", sItoA);
	}
	else if(BrbStringGetAdrOf(pText, "h", 0) != 0)
	{
		brsitoa((DINT)DtStruct.hour, (UDINT)&sItoA);
		BrbStringReplace(pText, "h", sItoA);
	}
	if(BrbStringGetAdrOf(pText, "MM", 0) != 0)
	{
		brsitoa((DINT)DtStruct.minute, (UDINT)&sItoA);
		if(DtStruct.minute < 10)
		{
			BrbStringInsert(sItoA, 0, "0");
		}
		BrbStringReplace(pText, "MM", sItoA);
	}
	else if(BrbStringGetAdrOf(pText, "M", 0) != 0)
	{
		brsitoa((DINT)DtStruct.minute, (UDINT)&sItoA);
		BrbStringReplace(pText, "M", sItoA);
	}
	if(BrbStringGetAdrOf(pText, "ss", 0) != 0)
	{
		brsitoa((DINT)DtStruct.second, (UDINT)&sItoA);
		if(DtStruct.second < 10)
		{
			BrbStringInsert(sItoA, 0, "0");
		}
		BrbStringReplace(pText, "ss", sItoA);
	}
	else if(BrbStringGetAdrOf(pText, "s", 0) != 0)
	{
		brsitoa((DINT)DtStruct.second, (UDINT)&sItoA);
		BrbStringReplace(pText, "s", sItoA);
	}
	return eBRB_ERR_OK;
}

// NOLINTEND(readability-*, bugprone-easily-swappable-parameters, bugprone-branch-clone, clang-diagnostic-invalid-utf8, clang-diagnostic-invalid-source-encoding, clang-diagnostic-pointer-arith, clang-diagnostic-strict-prototypes, hicpp-uppercase-literal-suffix, cppcoreguidelines-*, performance-*)
```

#### BrbUaGetRandomTimeZone.c
```c
#include <bur/plctypes.h>
#ifdef __cplusplus
	extern "C"
	{
#endif

#include "BrbLibUa.h"

#ifdef __cplusplus
	};
#endif

// NOLINTBEGIN(readability-*, bugprone-easily-swappable-parameters, bugprone-branch-clone, clang-diagnostic-invalid-utf8, clang-diagnostic-invalid-source-encoding, clang-diagnostic-pointer-arith, clang-diagnostic-strict-prototypes, hicpp-uppercase-literal-suffix, cppcoreguidelines-*, performance-*)

/* Erzeugt eine zufällige TimeZone */
plcdword BrbUaGetRandomTimeZone(BrUaTimeZoneDataType* pTimeZone)
{
	DWORD nStatus = 0x80460000; // = Bad_StructureMissing
	if(pTimeZone != 0)
	{
		nStatus = 0x00000000; // = Good
		pTimeZone->TimeOffset = (INT)BrbGetRandomDint(-12,12);
		pTimeZone->DaylightSaving = BrbGetRandomBool();
	}
	return nStatus;
}

// NOLINTEND(readability-*, bugprone-easily-swappable-parameters, bugprone-branch-clone, clang-diagnostic-invalid-utf8, clang-diagnostic-invalid-source-encoding, clang-diagnostic-pointer-arith, clang-diagnostic-strict-prototypes, hicpp-uppercase-literal-suffix, cppcoreguidelines-*, performance-*)
```

#### BrbUaGetRandomGuidString.c
```c
#include <bur/plctypes.h>
#ifdef __cplusplus
	extern "C"
	{
#endif

#include "BrbLibUa.h"
#include <string.h>

#ifdef __cplusplus
	};
#endif

// NOLINTBEGIN(readability-*, bugprone-easily-swappable-parameters, bugprone-branch-clone, clang-diagnostic-invalid-utf8, clang-diagnostic-invalid-source-encoding, clang-diagnostic-pointer-arith, clang-diagnostic-strict-prototypes, hicpp-uppercase-literal-suffix, cppcoreguidelines-*, performance-*)

/* Erzeugt einen zufälligen GuidString im Format '01234567-0123-0123-0123-0123456789AB' */
plcdword BrbUaGetRandomGuidString(BrUaGuidString* pGuidString, unsigned long nGuidStringSize, plcbit bWithSeparator)
{
	DWORD nStatus = 0x80460000; // = Bad_StructureMissing
	if(pGuidString != 0)
	{
		nStatus = 0x00000000; // = Good
		STRING sSelection[64];
		BrbStringCopy(sSelection, "0123456789abcdef", sizeof(sSelection));
		STRING sGuidStringElement[13];
		BrbGetRandomStringExt(sGuidStringElement, sizeof(sGuidStringElement), 8, sSelection);
		BrbStringCopy((STRING*)pGuidString, sGuidStringElement, nGuidStringSize);
		if(bWithSeparator == 1)
		{
			BrbStringCat((STRING*)pGuidString, "-", nGuidStringSize);
		}
		BrbGetRandomStringExt(sGuidStringElement, sizeof(sGuidStringElement), 4, sSelection);
		BrbStringCat((STRING*)pGuidString, sGuidStringElement, nGuidStringSize);
		if(bWithSeparator == 1)
		{
			BrbStringCat((STRING*)pGuidString, "-", nGuidStringSize);
		}
		BrbGetRandomStringExt(sGuidStringElement, sizeof(sGuidStringElement), 4, sSelection);
		BrbStringCat((STRING*)pGuidString, sGuidStringElement, nGuidStringSize);
		if(bWithSeparator == 1)
		{
			BrbStringCat((STRING*)pGuidString, "-", nGuidStringSize);
		}
		BrbGetRandomStringExt(sGuidStringElement, sizeof(sGuidStringElement), 4, sSelection);
		BrbStringCat((STRING*)pGuidString, sGuidStringElement, nGuidStringSize);
		if(bWithSeparator == 1)
		{
			BrbStringCat((STRING*)pGuidString, "-", nGuidStringSize);
		}
		BrbGetRandomStringExt(sGuidStringElement, sizeof(sGuidStringElement), 12, sSelection);
		BrbStringCat((STRING*)pGuidString, sGuidStringElement, nGuidStringSize);

	}
	return nStatus;
}

// NOLINTEND(readability-*, bugprone-easily-swappable-parameters, bugprone-branch-clone, clang-diagnostic-invalid-utf8, clang-diagnostic-invalid-source-encoding, clang-diagnostic-pointer-arith, clang-diagnostic-strict-prototypes, hicpp-uppercase-literal-suffix, cppcoreguidelines-*, performance-*)
```

#### BrbUaGetRandomXmlElement.c
```c
#include <bur/plctypes.h>
#ifdef __cplusplus
	extern "C"
	{
#endif
	#include "BrbLibUa.h"
#ifdef __cplusplus
	};
#endif

#include <string.h>

// NOLINTBEGIN(readability-*, bugprone-easily-swappable-parameters, bugprone-branch-clone, clang-diagnostic-invalid-utf8, clang-diagnostic-invalid-source-encoding, clang-diagnostic-pointer-arith, clang-diagnostic-strict-prototypes, hicpp-uppercase-literal-suffix, cppcoreguidelines-*, performance-*)

/* Erzeugt ein zufälliges XmlElement im Format '<Tag Attribute="X">Value</Tag>' */
plcdword BrbUaGetRandomXmlElement(BrUaXmlElement* pXmlElement)
{
	DWORD nStatus = 0x80460000; // = Bad_StructureMissing
	if(pXmlElement != 0)
	{
		nStatus = 0x00000000; // = Good
		BrbStringCopy(pXmlElement->Data, "<Tag Attribute=", sizeof(pXmlElement->Data));
		BrbStringCat(pXmlElement->Data, (STRING*)&sBRB_QM, sizeof(pXmlElement->Data));
		UDINT nNumber = (UDINT)BrbGetRandomDint(0, 255);
		STRING sNumber[12];
		brsitoa((DINT)nNumber, (UDINT)&sNumber);
		BrbStringCat(pXmlElement->Data, sNumber, sizeof(pXmlElement->Data));
		BrbStringCat(pXmlElement->Data, (STRING*)&sBRB_QM, sizeof(pXmlElement->Data));
		BrbStringCat(pXmlElement->Data, ">Value</Tag>", sizeof(pXmlElement->Data));
		pXmlElement->Length = (DINT)strlen((STRING*)&pXmlElement->Data);
	}
	return nStatus;
}

// NOLINTEND(readability-*, bugprone-easily-swappable-parameters, bugprone-branch-clone, clang-diagnostic-invalid-utf8, clang-diagnostic-invalid-source-encoding, clang-diagnostic-pointer-arith, clang-diagnostic-strict-prototypes, hicpp-uppercase-literal-suffix, cppcoreguidelines-*, performance-*)
```

#### Package Logical/Libraries/BrbLibUa/Client/Connection - Funktionen für OpcUa-Verbindungen

#### BrbUaGetConnectionStatusText.c
```c
#include <bur/plctypes.h>
#ifdef __cplusplus
	extern "C"
	{
#endif

#include "BrbLibUa.h"
#include <string.h>

#ifdef __cplusplus
	};
#endif

// NOLINTBEGIN(readability-*, bugprone-easily-swappable-parameters, bugprone-branch-clone, clang-diagnostic-invalid-utf8, clang-diagnostic-invalid-source-encoding, clang-diagnostic-pointer-arith, clang-diagnostic-strict-prototypes, hicpp-uppercase-literal-suffix, cppcoreguidelines-*, performance-*)

/* Gibt einen Verbindungs-Status als Text zurück */
plcdword BrbUaGetConnectionStatusText(enum UAConnectionStatus eConnectionStatus, plcstring* pStatusText, unsigned long nStatusTextSize)
{
	DWORD nStatus = 0x80460000; // = Bad_StructureMissing
	if(pStatusText != 0)
	{
		nStatus = 0x00000000; // = Good
		memset(pStatusText, 0, nStatusTextSize);
		switch(eConnectionStatus) // NOLINT(hicpp-multiway-paths-covered)
		{
			case UACS_Connected:
				BrbStringCopy(pStatusText, "Connected", nStatusTextSize);
				break;

			case UACS_ConnectionError:
				BrbStringCopy(pStatusText, "ConnectionError", nStatusTextSize);
				break;

			case UACS_Shutdown:
				BrbStringCopy(pStatusText, "Shutdown", nStatusTextSize);
				break;
		}
	}
	return nStatus;
}

// NOLINTEND(readability-*, bugprone-easily-swappable-parameters, bugprone-branch-clone, clang-diagnostic-invalid-utf8, clang-diagnostic-invalid-source-encoding, clang-diagnostic-pointer-arith, clang-diagnostic-strict-prototypes, hicpp-uppercase-literal-suffix, cppcoreguidelines-*, performance-*)
```
